% RSLogix 500 project PROJECT7.RSS, saved by version 8.30.00.16 %
PROJECT "PRO7"    % processor: Bul.1763 MicroLogix 1100 Series B %

PROGRAM FILES
  LAD 2 "MAIN"  4 rungs
  LAD 3 "IO"  3 rungs
  LAD 4 "VALVE CTRL"  8 rungs
  LAD 5 "CALIBRATE"  9 rungs

DATA FILES
  O0 OUTPUT  4 elements
  I1 INPUT  6 elements
  S2 STATUS  66 elements
  B3 BINARY  1 elements
  T4 TIMER  5 elements
  C5 COUNTER  2 elements
  R6 CONTROL  1 elements
  N7 INTEGER  11 elements
  F8 FLOAT  7 elements

LADDER 2 "MAIN"
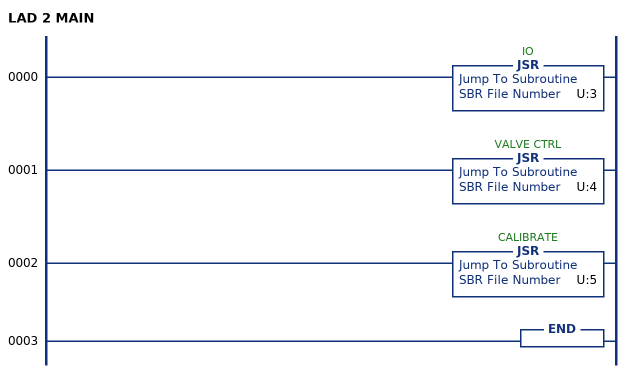
% Rung: 0 %
SOR JSR U:3 EOR
%   U:3  "IO" %
% Rung: 1 %
SOR JSR U:4 EOR
%   U:4  "VALVE CTRL" %
% Rung: 2 %
SOR JSR U:5 EOR
%   U:5  "CALIBRATE" %
% Rung: 3 %
SOR END EOR

LADDER 3 "IO"
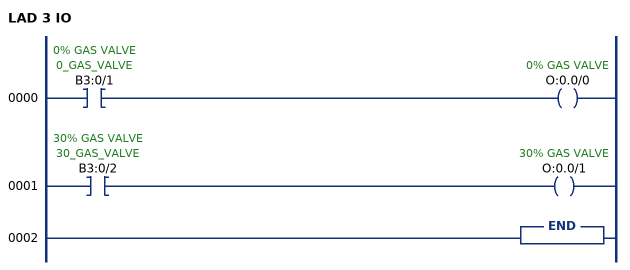
% Rung: 0 %
SOR XIC B3:0/1 OTE O:0.0/0 EOR
%   B3:0/1  0_GAS_VALVE  "0% GAS VALVE" %
%   O:0.0/0  "0% GAS VALVE" %
% Rung: 1 %
SOR XIC B3:0/2 OTE O:0.0/1 EOR
%   B3:0/2  30_GAS_VALVE  "30% GAS VALVE" %
%   O:0.0/1  "30% GAS VALVE" %
% Rung: 2 %
SOR END EOR

LADDER 4 "VALVE CTRL"
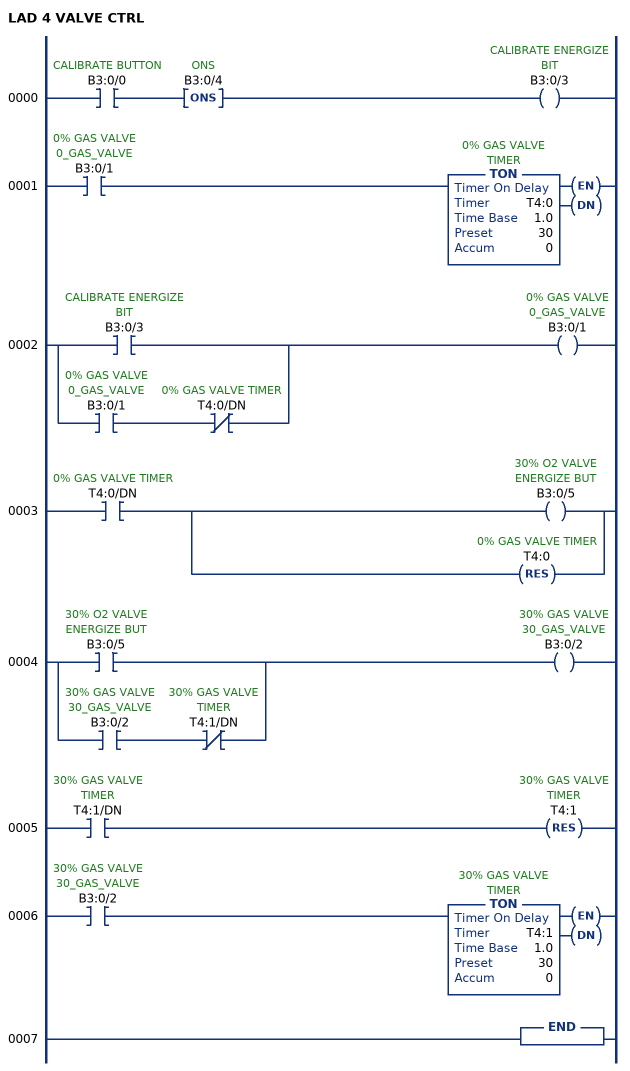
% Rung: 0 %
SOR XIC B3:0/0 ONS B3:0/4 OTE B3:0/3 EOR
%   B3:0/0  "CALIBRATE BUTTON" %
%   B3:0/4  "ONS" %
%   B3:0/3  "CALIBRATE ENERGIZE BIT" %
% Rung: 1 %
SOR XIC B3:0/1 TON T4:0 1.0 30 0 EOR
%   B3:0/1  0_GAS_VALVE  "0% GAS VALVE" %
%   T4:0  "0% GAS VALVE TIMER" %
% Rung: 2 %
SOR BST XIC B3:0/3 NXB XIC B3:0/1 XIO T4:0/DN BND OTE B3:0/1 EOR
%   B3:0/3  "CALIBRATE ENERGIZE BIT" %
%   B3:0/1  0_GAS_VALVE  "0% GAS VALVE" %
%   T4:0  "0% GAS VALVE TIMER" %
% Rung: 3 %
SOR XIC T4:0/DN BST OTE B3:0/5 NXB RES T4:0 BND EOR
%   T4:0  "0% GAS VALVE TIMER" %
%   B3:0/5  "30% O2 VALVE ENERGIZE BUT" %
% Rung: 4 %
SOR BST XIC B3:0/5 NXB XIC B3:0/2 XIO T4:1/DN BND OTE B3:0/2 EOR
%   B3:0/5  "30% O2 VALVE ENERGIZE BUT" %
%   B3:0/2  30_GAS_VALVE  "30% GAS VALVE" %
%   T4:1  "30% GAS VALVE TIMER" %
% Rung: 5 %
SOR XIC T4:1/DN RES T4:1 EOR
%   T4:1  "30% GAS VALVE TIMER" %
% Rung: 6 %
SOR XIC B3:0/2 TON T4:1 1.0 30 0 EOR
%   B3:0/2  30_GAS_VALVE  "30% GAS VALVE" %
%   T4:1  "30% GAS VALVE TIMER" %
% Rung: 7 %
SOR END EOR

LADDER 5 "CALIBRATE"
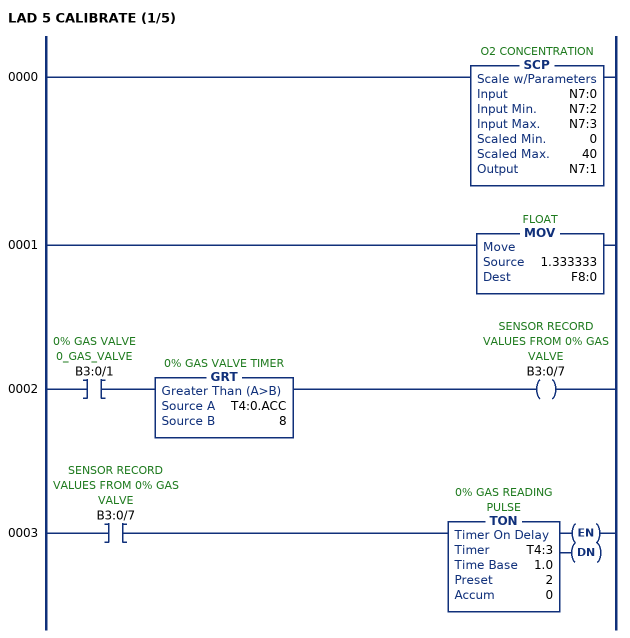
% Rung: 0 %
SOR SCP N7:0 N7:2 N7:3 0 40 N7:1 EOR
%   N7:0  "O2 INPUT SIGNAL" %
%   N7:2  "INPUT MIN" %
%   N7:3  "INPUT MAX" %
%   N7:1  "O2 CONCENTRATION" %
% Rung: 1 %
SOR MOV 1.333333 F8:0 EOR
%   F8:0  "FLOAT" %
% Rung: 2 %
SOR XIC B3:0/1 GRT T4:0.ACC 8 OTE B3:0/7 EOR
%   B3:0/1  0_GAS_VALVE  "0% GAS VALVE" %
%   T4:0  "0% GAS VALVE TIMER" %
%   B3:0/7  "SENSOR RECORD VALUES FROM 0% GAS VALVE" %
% Rung: 3 %
SOR XIC B3:0/7 TON T4:3 1.0 2 0 EOR
%   B3:0/7  "SENSOR RECORD VALUES FROM 0% GAS VALVE" %
%   T4:3  "0% GAS READING PULSE" %

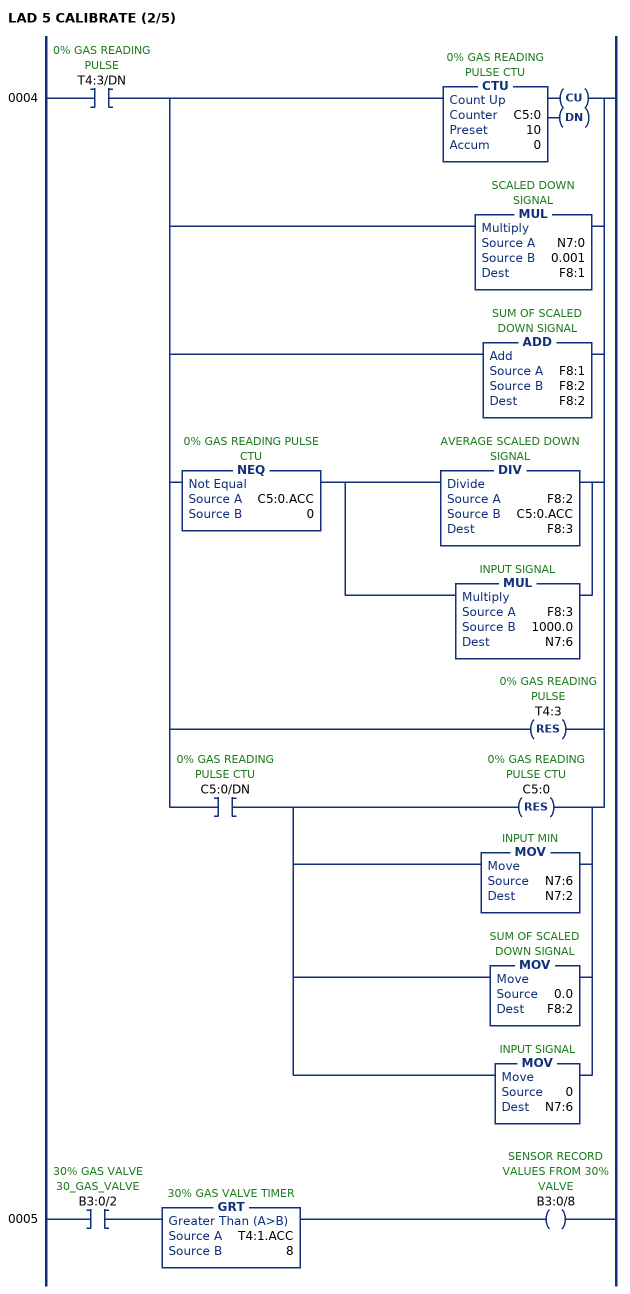
% Rung: 4 %
SOR XIC T4:3/DN BST CTU C5:0 10 0 NXB MUL N7:0 0.001 F8:1 NXB ADD F8:1 F8:2 F8:2 NXB NEQ C5:0.ACC 0 BST DIV F8:2 C5:0.ACC F8:3 NXB MUL F8:3 1000.0 N7:6 BND NXB RES T4:3 NXB XIC C5:0/DN BST RES C5:0 NXB MOV N7:6 N7:2 NXB MOV 0.0 F8:2 NXB MOV 0 N7:6 BND BND EOR
%   T4:3  "0% GAS READING PULSE" %
%   C5:0  "0% GAS READING PULSE CTU" %
%   N7:0  "O2 INPUT SIGNAL" %
%   F8:1  "SCALED DOWN SIGNAL" %
%   F8:2  "SUM OF SCALED DOWN SIGNAL" %
%   F8:3  "AVERAGE SCALED DOWN SIGNAL" %
%   N7:6  "INPUT SIGNAL" %
%   N7:2  "INPUT MIN" %
% Rung: 5 %
SOR XIC B3:0/2 GRT T4:1.ACC 8 OTE B3:0/8 EOR
%   B3:0/2  30_GAS_VALVE  "30% GAS VALVE" %
%   T4:1  "30% GAS VALVE TIMER" %
%   B3:0/8  "SENSOR RECORD VALUES FROM 30% VALVE" %

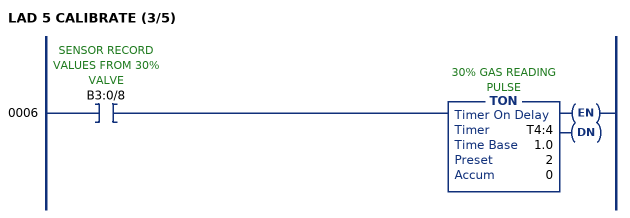
% Rung: 6 %
SOR XIC B3:0/8 TON T4:4 1.0 2 0 EOR
%   B3:0/8  "SENSOR RECORD VALUES FROM 30% VALVE" %
%   T4:4  "30% GAS READING PULSE" %

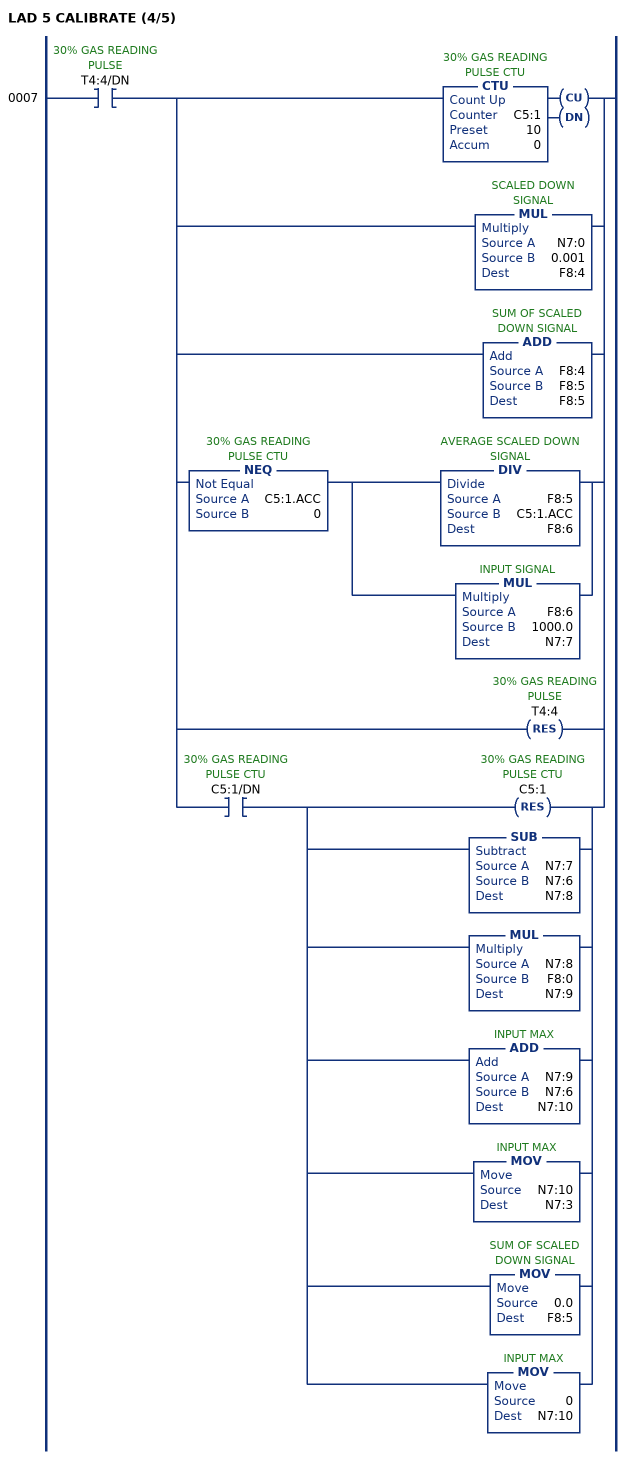
% Rung: 7 %
SOR XIC T4:4/DN BST CTU C5:1 10 0 NXB MUL N7:0 0.001 F8:4 NXB ADD F8:4 F8:5 F8:5 NXB NEQ C5:1.ACC 0 BST DIV F8:5 C5:1.ACC F8:6 NXB MUL F8:6 1000.0 N7:7 BND NXB RES T4:4 NXB XIC C5:1/DN BST RES C5:1 NXB SUB N7:7 N7:6 N7:8 NXB MUL N7:8 F8:0 N7:9 NXB ADD N7:9 N7:6 N7:10 NXB MOV N7:10 N7:3 NXB MOV 0.0 F8:5 NXB MOV 0 N7:10 BND BND EOR
%   T4:4  "30% GAS READING PULSE" %
%   C5:1  "30% GAS READING PULSE CTU" %
%   N7:0  "O2 INPUT SIGNAL" %
%   F8:4  "SCALED DOWN SIGNAL" %
%   F8:5  "SUM OF SCALED DOWN SIGNAL" %
%   F8:6  "AVERAGE SCALED DOWN SIGNAL" %
%   N7:7  "INPUT SIGNAL" %
%   N7:6  "INPUT SIGNAL" %
%   F8:0  "FLOAT" %
%   N7:10  "INPUT MAX" %
%   N7:3  "INPUT MAX" %

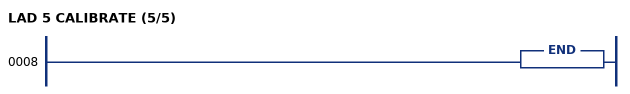
% Rung: 8 %
SOR END EOR

OTHER DOCUMENTED ADDRESSES
  F8:7  "AVERAGE SIGNAL"

DATA TABLE (non-zero values as saved)
DATA T4
% .PRE .ACC %
% T4:0 % 30 0
% T4:1 % 30 0
% T4:3 % 2 0
% T4:4 % 2 0
DATA C5
% .PRE .ACC %
% C5:0 % 10 0
% C5:1 % 10 0
DATA N7
% N7:0 % 0 0 0 16383 0 0 0 0 0 0
